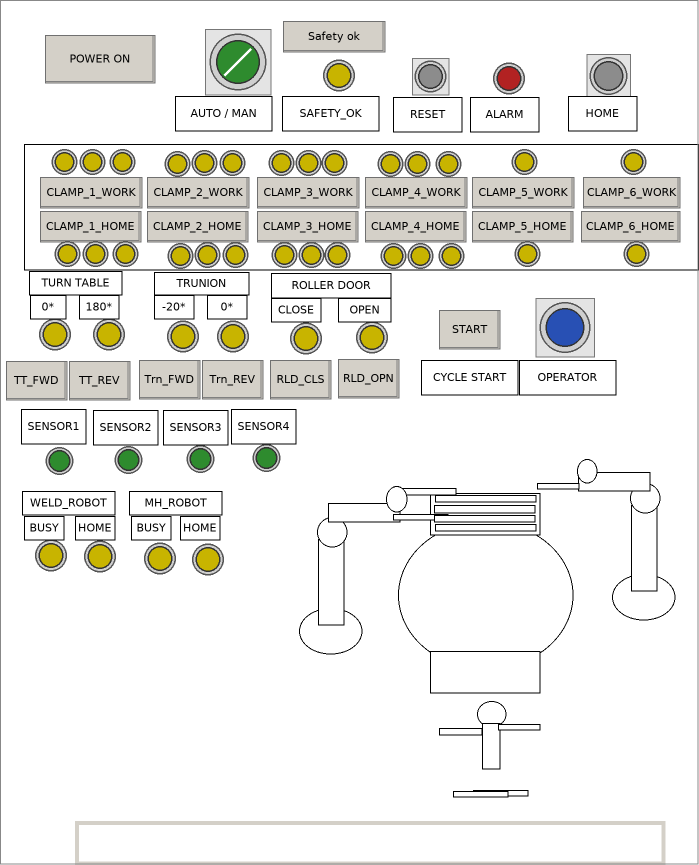
VISUALIZATION AUTO_PROCESS  // 699x865
    Rectangle (24,144 675x126)
    Lamp1 (314,57 50x37), variable: OP_Memory_DB.SAFETY_OK, style: Lamp-Lamp1-Yellow
    RotarySwitch (205,23 66x78), variable: OP_Memory_DB.Auto_mode, behaviour: TOGGLE, style: Switch-RotarySwitch-Green
    Rectangle (175,96 97x35), "AUTO / MAN"
    Rectangle (393,97 69x35), "RESET"
    Button (45,35 110x48), "POWER ON", colour toggle: OP_Memory_DB.POWER_ON
        toggle OP_Memory_DB.POWER_ON
    Button (40,177 102x31), "CLAMP_1_WORK", colour toggle: OP_Memory_DB.M_CC1_CLAMPING_UNIT1_3_WP
        toggle OP_Memory_DB.M_CC1_CLAMPING_UNIT1_3_WP
    Button (40,211 101x31), "CLAMP_1_HOME", colour toggle: OP_Memory_DB.M_CC1_CLAMPING_UNIT1_3_HP
        toggle OP_Memory_DB.M_CC1_CLAMPING_UNIT1_3_HP
    Button (583,177 97x31), "CLAMP_6_WORK", colour toggle: OP_Memory_DB.M_CC6_CLAMPING_UNIT6_1_WP
        toggle OP_Memory_DB.M_CC6_CLAMPING_UNIT6_1_WP
    Button (472,177 102x31), "CLAMP_5_WORK", colour toggle: OP_Memory_DB.M_CC5_CLAMPING_UNIT5_1_WP
        toggle OP_Memory_DB.M_CC5_CLAMPING_UNIT5_1_WP
    Button (472,211 101x31), "CLAMP_5_HOME", colour toggle: OP_Memory_DB.M_CC5_CLAMPING_UNIT5_1_HP
        toggle OP_Memory_DB.M_CC5_CLAMPING_UNIT5_1_HP
    Button (581,211 99x31), "CLAMP_6_HOME", colour toggle: OP_Memory_DB.M_CC6_CLAMPING_UNIT6_1_HP
        toggle OP_Memory_DB.M_CC6_CLAMPING_UNIT6_1_HP
    Rectangle (29,271 93x24), "TURN TABLE"
    Rectangle (154,272 95x23), "TRUNION"
    Rectangle (271,273 120x25), "ROLLER DOOR"
    Lamp1 (30,316 50x37), variable: Inputs.i_1st_TT_Pos, style: Lamp-Lamp1-Yellow
    Lamp1 (84,316 50x37), variable: Inputs.i_2nd_TT_Pos, style: Lamp-Lamp1-Yellow
    Lamp1 (158,318 50x37), variable: Inputs.i_Trunion_1st_Pos, style: Lamp-Lamp1-Yellow
    Lamp1 (208,318 50x37), variable: Inputs.i_Trunion_2nd_Pos, style: Lamp-Lamp1-Yellow
    Lamp1 (281,320 50x37), variable: Inputs.i_ROLL_DR_Close_Pos_LS, style: Lamp-Lamp1-Yellow
    Lamp1 (347,319 50x37), variable: Inputs.i_ROLL_DR_Open_Pos_LS, style: Lamp-Lamp1-Yellow
    Button (147,177 102x31), "CLAMP_2_WORK", colour toggle: OP_Memory_DB.M_CC2_CLAMPING_UNIT2_3_WP
        toggle OP_Memory_DB.M_CC2_CLAMPING_UNIT2_3_WP
    Button (147,211 101x31), "CLAMP_2_HOME", colour toggle: OP_Memory_DB.M_CC2_CLAMPING_UNIT2_3_HP
        toggle OP_Memory_DB.M_CC2_CLAMPING_UNIT2_3_HP
    Button (257,177 102x31), "CLAMP_3_WORK", colour toggle: OP_Memory_DB.M_CC3_CLAMPING_UNIT3_3_WP
        toggle OP_Memory_DB.M_CC3_CLAMPING_UNIT3_3_WP
    Button (257,211 101x31), "CLAMP_3_HOME", colour toggle: OP_Memory_DB.M_CC3_CLAMPING_UNIT3_3_HP
        toggle OP_Memory_DB.M_CC3_CLAMPING_UNIT3_3_HP
    Button (365,177 102x31), "CLAMP_4_WORK", colour toggle: OP_Memory_DB.M_CC4_CLAMPING_UNIT4_3_WP
        toggle OP_Memory_DB.M_CC4_CLAMPING_UNIT4_3_WP
    Button (365,211 101x31), "CLAMP_4_HOME", colour toggle: OP_Memory_DB.M_CC4_CLAMPING_UNIT4_3_HP
        toggle OP_Memory_DB.M_CC4_CLAMPING_UNIT4_3_HP
    Rectangle (30,295 36x24), "0*"
    Rectangle (79,295 40x24), "180*"
    Rectangle (154,295 40x24), "-20*"
    Rectangle (207,295 40x24), "0*"
    Rectangle (271,298 50x24), "CLOSE"
    Rectangle (338,298 53x24), "OPEN"
    Button (6,361 61x39), "TT_FWD", colour toggle: OP_Memory_DB.M_2ND_POSITION_TT_CMD
        tap OP_Memory_DB.M_2ND_POSITION_TT_CMD
    Button (69,361 61x39), "TT_REV", colour toggle: OP_Memory_DB.M_1ST_POSITION_TT_CMD
        tap OP_Memory_DB.M_1ST_POSITION_TT_CMD
    Button (139,360 61x39), "Trn_FWD", colour toggle: OP_Memory_DB.M_Fwd_POSITION
        tap OP_Memory_DB.M_Fwd_POSITION
    Button (202,360 61x39), "Trn_REV", colour toggle: OP_Memory_DB.M_Rev_POSITION
        tap OP_Memory_DB.M_Rev_POSITION
    Button (338,359 61x39), "RLD_OPN", colour toggle: OP_Memory_DB.M_Roll_Dr_Open
        tap OP_Memory_DB.M_Roll_Dr_Open
    Button (270,360 61x39), "RLD_CLS", colour toggle: OP_Memory_DB.M_Roll_Dr_Close
        tap OP_Memory_DB.M_Roll_Dr_Close
    PushSwitch (535,298 60x59), variable: Inputs.i_OPERATE_START_PB, behaviour: TAP, style: Switch-PushSwitch-Blue
    Rectangle (519,360 97x35), "OPERATOR"
    Rectangle (21,409 65x35), "SENSOR1"
    Lamp1 (178,443 45x32), variable: Inputs.i_PART_CONTROL_B8, style: Lamp-Lamp1-Green
    Lamp1 (247,442 39x32), variable: Inputs.i_PART_CONTROL_B22, style: Lamp-Lamp1-Green
    Rectangle (93,410 65x35), "SENSOR2"
    Rectangle (163,410 65x35), "SENSOR3"
    Rectangle (231,409 65x35), "SENSOR4"
    Lamp1 (37,445 45x32), variable: Inputs.i_PART_CONTROL_B1, style: Lamp-Lamp1-Green
    Lamp1 (106,444 45x32), variable: Inputs.i_PART_CONTROL_B15, style: Lamp-Lamp1-Green
    Ellipse (398,521 175x148)
    Rectangle (430,493 110x42)
    Rectangle (430,651 110x42)
    Ellipse (612,574 63x46)
    Rectangle (631,505 26x86)
    Ellipse (630,483 30x30)
    Rectangle (578,472 72x19), angle 26
    Rectangle (537,483 42x6), angle 337, colour toggle: OP_Memory_DB.ROBOT_BUSY
    Ellipse (299,608 63x46)
    Rectangle (318,539 26x86)
    Ellipse (317,517 30x30)
    Rectangle (328,503 72x19), angle 335
    Rectangle (399,488 57x7), angle 349, colour toggle: OP_Memory_DB.MH_ROBOT_BUSY
    Rectangle (393,514 55x6), angle 54, colour toggle: OP_Memory_DB.MH_ROBOT_BUSY
    Ellipse (577,459 20x24)
    Ellipse (386,486 21x26)
    Ellipse (477,701 29x26)
    Rectangle (482,723 18x46)
    Rectangle (498,724 42x6), angle 337, colour toggle: Inputs.i_OPERATE_START_PB
    Rectangle (473,790 55x6), angle 69
    Rectangle (453,791 55x6), angle 111
    Rectangle (439,728 43x7), angle 9, colour toggle: Inputs.i_OPERATE_START_PB
    Lamp1 (45,147 39x30), variable: Inputs.i_CC1_Clamp_1_Sensor_WP, style: Lamp-Lamp1-Yellow
    PushSwitch (409,58 43x37), variable: Inputs.i_Reset_PB, behaviour: TAP, style: Switch-PushSwitch-Gray
    Rectangle (282,96 97x35), "SAFETY_OK"
    Lamp1 (484,60 50x37), variable: Outputs.O_FAULT_LAMP, style: Lamp-Lamp1-Red
    Rectangle (470,97 69x35), "ALARM"
    Lamp1 (158,149 39x30), variable: Inputs.i_CC2_Clamp_1_Sensor_WP, style: Lamp-Lamp1-Yellow
    Lamp1 (262,148 39x30), variable: Inputs.i_CC3_Clamp_1_Sensor_WP, style: Lamp-Lamp1-Yellow
    Lamp1 (371,149 39x30), variable: Inputs.i_CC4_Clamp_1_Sensor_WP, style: Lamp-Lamp1-Yellow
    Lamp1 (505,147 39x30), variable: Inputs.i_CC5_Clamp_1_Sensor_WP, style: Lamp-Lamp1-Yellow
    Lamp1 (614,147 39x30), variable: Inputs.i_CC6_Clamp_1_Sensor_WP, style: Lamp-Lamp1-Yellow
    PushSwitch (580,54 57x44), variable: OP_Memory_DB.M_FIX1_ALL_CLAMP_HOME_PB, behaviour: TAP, style: Switch-PushSwitch-Gray
    Rectangle (568,96 69x35), "HOME"
    Lamp1 (73,147 39x30), variable: Inputs.i_CC1_Clamp_2_Sensor_WP, style: Lamp-Lamp1-Yellow
    Lamp1 (103,147 39x30), variable: Inputs.i_CC1_Clamp_3_Sensor_WP, style: Lamp-Lamp1-Yellow
    Lamp1 (185,148 39x30), variable: Inputs.i_CC2_Clamp_2_Sensor_WP, style: Lamp-Lamp1-Yellow
    Lamp1 (213,148 39x30), variable: Inputs.i_CC2_Clamp_3_Sensor_WP, style: Lamp-Lamp1-Yellow
    Lamp1 (289,148 39x30), variable: Inputs.i_CC3_Clamp_2_Sensor_WP, style: Lamp-Lamp1-Yellow
    Lamp1 (315,148 39x30), variable: Inputs.i_CC3_Clamp_3_Sensor_WP, style: Lamp-Lamp1-Yellow
    Lamp1 (398,149 39x30), variable: Inputs.i_CC4_Clamp_2_Sensor_WP, style: Lamp-Lamp1-Yellow
    Lamp1 (429,149 39x30), variable: Inputs.i_CC4_Clamp_3_Sensor_WP, style: Lamp-Lamp1-Yellow
    Button (283,21 102x31), "Safety ok", colour toggle: OP_Memory_DB.SAFETY_OK
        toggle OP_Memory_DB.SAFETY_OK
    Rectangle (421,360 97x35), "CYCLE START"
    Lamp1 (48,239 39x30), variable: Inputs.i_CC1_Clamp_1_Sensor_HP, style: Lamp-Lamp1-Yellow
    Lamp1 (161,241 39x30), variable: Inputs.i_CC2_Clamp_1_Sensor_HP, style: Lamp-Lamp1-Yellow
    Lamp1 (265,240 39x30), variable: Inputs.i_CC3_Clamp_1_Sensor_HP, style: Lamp-Lamp1-Yellow
    Lamp1 (374,241 39x30), variable: Inputs.i_CC4_Clamp_1_Sensor_HP, style: Lamp-Lamp1-Yellow
    Lamp1 (508,239 39x30), variable: Inputs.i_CC5_Clamp_1_Sensor_HP, style: Lamp-Lamp1-Yellow
    Lamp1 (617,239 39x30), variable: Inputs.i_CC6_Clamp_1_Sensor_HP, style: Lamp-Lamp1-Yellow
    Lamp1 (76,239 39x30), variable: Inputs.i_CC1_Clamp_2_Sensor_HP, style: Lamp-Lamp1-Yellow
    Lamp1 (106,239 39x30), variable: Inputs.i_CC1_Clamp_3_Sensor_HP, style: Lamp-Lamp1-Yellow
    Lamp1 (188,240 39x30), variable: Inputs.i_CC2_Clamp_2_Sensor_HP, style: Lamp-Lamp1-Yellow
    Lamp1 (216,240 39x30), variable: Inputs.i_CC2_Clamp_3_Sensor_HP, style: Lamp-Lamp1-Yellow
    Lamp1 (292,240 39x30), variable: Inputs.i_CC3_Clamp_2_Sensor_HP, style: Lamp-Lamp1-Yellow
    Lamp1 (318,240 39x30), variable: Inputs.i_CC3_Clamp_3_Sensor_HP, style: Lamp-Lamp1-Yellow
    Lamp1 (401,241 39x30), variable: Inputs.i_CC4_Clamp_2_Sensor_HP, style: Lamp-Lamp1-Yellow
    Lamp1 (432,241 39x30), variable: Inputs.i_CC4_Clamp_3_Sensor_HP, style: Lamp-Lamp1-Yellow
    Button (439,310 61x39), "START", colour toggle: Inputs.i_CYCLE_START_PB
        tap Inputs.i_CYCLE_START_PB
    Rectangle (22,491 93x24), "WELD_ROBOT"
    Lamp1 (135,540 50x37), variable: OP_Memory_DB.MH_ROBOT_BUSY, style: Lamp-Lamp1-Yellow
    Lamp1 (183,541 50x37), variable: OP_Memory_DB.MH_ROBOT_HOME, style: Lamp-Lamp1-Yellow
    Rectangle (129,491 93x24), "MH_ROBOT"
    Lamp1 (26,537 50x37), variable: OP_Memory_DB.ROBOT_BUSY, style: Lamp-Lamp1-Yellow
    Lamp1 (75,538 50x37), variable: OP_Memory_DB.ROBOT_HOME, style: Lamp-Lamp1-Yellow
    Rectangle (24,516 40x24), "BUSY"
    Rectangle (75,516 40x24), "HOME"
    Rectangle (131,516 40x24), "BUSY"
    Rectangle (180,516 40x24), "HOME"
    Textfield (75,821 590x44), text list: 'FiX_1', text index: BLOCK_CALL.MODE_CONTROL_DB.Step
    Rectangle (435,495 101x7), colour toggle: Inputs.i_PART_CONTROL_B1
    Rectangle (434,505 101x8), colour toggle: Inputs.i_PART_CONTROL_B15
    Rectangle (434,515 101x7), colour toggle: Inputs.i_PART_CONTROL_B8
    Rectangle (435,524 101x7), colour toggle: Inputs.i_PART_CONTROL_B22
END_VISUALIZATION

(* stored: Version 1.1.0.1, ProductVersion 3.1.4024.16
   Visu AUTO_PROCESS: Id {7d852165-6a8a-4da3-b035-ec4b3b6b2056} *)
